# EPICS substitutions: iocBoot/ioc13MeasComp2408_2/pid_slow.substitutions
file "$(STD)/db/pid_control.db"
{
pattern
{P,            PID,        INP,             OUT,         LOPR,  HOPR,  DRVL,  DRVH,  PREC,   KP,  KI,   KD,  SCAN}
{13USB2408_2:, PID1, 13USB2408_2:Ti1,  13USB2408_2:Ao1,   0,    100,     0,    5,     3,     0.2,  3.,   0.,  ".1 second"}
}
